FUNCTION_BLOCK FB_UAconnectMock_Success IMPLEMENTS I_OPCUA_Connect
VAR_INPUT
END_VAR
VAR_OUTPUT
END_VAR
VAR
END_VAR

{warning 'add method implementation '}
METHOD start : BOOL
VAR_INPUT
	Execute	: BOOL;
	ServerUrl	: STRING(MAX_STRING_LENGTH);
	SessionConnectInfo	: Tc3_PLCopen_OpcUa.ST_UASessionConnectInfo;
	Timeout	: TIME := DEFAULT_ADS_TIMEOUT;
END_VAR
VAR_OUTPUT
	ConnectionHdl	: DWORD;
	Done	: BOOL;
	Busy	: BOOL;
	Error	: BOOL;
	ErrorID	: DWORD;
END_VAR
IF execute THEN
	done := TRUE;
END_IF
END_METHOD

END_FUNCTION_BLOCK

(* stored: Version 1.1.0.1, ProductVersion 3.1.4024.9
   POU FB_UAconnectMock_Success: Id {8b7f916b-1dd5-4457-a43a-10e9e68a92ec}, SpecialFunc None
   Method start: Id {275e55f8-ee51-47ac-b6fb-7e9596ac938d} *)
